Staubli VAL3: TrajPoint.pjx

--- TrajPoint.pjx ---
Parameters version=s7.5 stackSize=5000 millimeterUnit=true
Data file=TrajPoint.dtx
Type name=TrajPointItem path=Disk://kernel/template/TrajPointItem/TrajPointItem.pjx

--- TrajPoint.dtx ---
public TrajPointItem tData[3]
  [0]
    TrajectoryItem tSuper
      [0]
        num distance
        num moveType
        num nTime
        num nStop
        num nTcpAction
        string comment
        bool toStop
        mdesc nom_speed = {vel=450, tmax=500, leave=30, reach=30}
        InstrItem iInstr[3]
          [0]
            string sType
            string sData
          [1]
            string sType
            string sData
          [2]
            string sType
            string sData
        num nMoveId
    pointRx pPoint = {fatherId=fFrame[0]}
    num nType
  [1]
    TrajectoryItem tSuper
      [0]
        num distance
        num moveType
        num nTime
        num nStop
        num nTcpAction
        string comment
        bool toStop
        mdesc nom_speed = {vel=450, tmax=1000, leave=30, reach=30, blend=off}
        InstrItem iInstr[3]
          [0]
            string sType
            string sData
          [1]
            string sType
            string sData
          [2]
            string sType
            string sData
        num nMoveId
    pointRx pPoint
    num nType
  [2]
    TrajectoryItem tSuper
      [0]
        num distance
        num moveType
        num nTime
        num nStop
        num nTcpAction
        string comment
        bool toStop
        mdesc nom_speed = {vel=450, tmax=500, leave=30, reach=30}
        InstrItem iInstr[3]
          [0]
            string sType
            string sData
          [1]
            string sType
            string sData
          [2]
            string sType
            string sData
        num nMoveId
    pointRx pPoint
    num nType
public frame fFrame = {fatherId=world[0]}
public num nIndexTool
public string sID
public num nIndexFrame
